SYSTEM System
  DEVICE EcoRT_0 : Soft_dPAC
    RESOURCE RES0 : EMB_RES_ECO
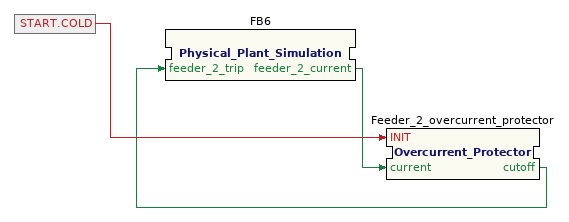
      FBS
        FB6 : Physical_Plant_Simulation;
        Feeder_2_overcurrent_protector : Overcurrent_Protector;
      END_FBS
      EVENT_CONNECTIONS
        START.COLD TO Feeder_2_overcurrent_protector.INIT;
      END_CONNECTIONS
      ADAPTER_CONNECTIONS
        FB6.feeder_2_current TO Feeder_2_overcurrent_protector.current;
        Feeder_2_overcurrent_protector.cutoff TO FB6.feeder_2_trip;
      END_CONNECTIONS
    END_RESOURCE
  END_DEVICE
END_SYSTEM
